// TIA Portal V20 export
DATA_BLOCK "InstShiftProductionTimes"   // DB113
TITLE = Instance ShiftProductionTimes
{ DB_Accessible_From_OPC_UA := 'FALSE' }
AUTHOR : SICAR
FAMILY : Shift
// Instance DB
// stored: DBAccessibleFromOPCUA false, InstanceOfName LSicar_ShiftProductionTimes, InstanceOfType FB
"LSicar_ShiftProductionTimes"
   // VAR_OUTPUT
   //    shiftProdTimeTarget { ExternalAccessible := 'False'; ExternalVisible := 'False'; ExternalWritable := 'False'} : Time := T#0MS;
   //    shiftProdTimeExpired { ExternalAccessible := 'False'; ExternalVisible := 'False'; ExternalWritable := 'False'} : Time := T#0MS;
   //    shiftActive { ExternalAccessible := 'False'; ExternalVisible := 'False'; ExternalWritable := 'False'} : Bool := FALSE;
   //    shiftFinishedPulse { ExternalAccessible := 'False'; ExternalVisible := 'False'; ExternalWritable := 'False'} : Bool := FALSE;
   // END_VAR
   // VAR_IN_OUT
   //    dateAndTime : "LSicar_typeGlobalDateTime";
   //    prodTimesHmi : "LSicar_typeProdTimesHmi";
   // END_VAR
   // VAR
   //    statCurrShiftTimes { ExternalAccessible := 'False'; ExternalVisible := 'False'; ExternalWritable := 'False'} : "LSicar_typeShiftTimes1Shift";
   //    statActual { ExternalAccessible := 'False'; ExternalVisible := 'False'; ExternalWritable := 'False'} : Time_Of_Day := TOD#00:00:00;
   //    statBefore { ExternalAccessible := 'False'; ExternalVisible := 'False'; ExternalWritable := 'False'} : Time_Of_Day := TOD#00:00:00;
   //    statDayChange { ExternalAccessible := 'False'; ExternalVisible := 'False'; ExternalWritable := 'False'} : Bool := FALSE;
   //    statDayChangeSet { ExternalAccessible := 'False'; ExternalVisible := 'False'; ExternalWritable := 'False'} : Bool := FALSE;
   //    statShift { ExternalAccessible := 'False'; ExternalVisible := 'False'; ExternalWritable := 'False'} : "LSicar_typeShiftmodelInfo";
   //    statProdTimeExpired { ExternalAccessible := 'False'; ExternalVisible := 'False'; ExternalWritable := 'False'} : Time := T#0MS;
   //    statBreak { ExternalAccessible := 'False'; ExternalVisible := 'False'; ExternalWritable := 'False'} : Array[0..4] of "LSicar_typeShiftmodelInfo";
   //    statBreakDurationSummary { ExternalAccessible := 'False'; ExternalVisible := 'False'; ExternalWritable := 'False'} : Time := T#0MS;
   //    statBreakActiveSummary { ExternalAccessible := 'False'; ExternalVisible := 'False'; ExternalWritable := 'False'} : Bool := FALSE;
   //    statBreakCount { ExternalAccessible := 'False'; ExternalVisible := 'False'; ExternalWritable := 'False'} : USInt := 0;
   //    statProdTimeExpired1 { ExternalAccessible := 'False'; ExternalVisible := 'False'; ExternalWritable := 'False'} : Time := T#0MS;
   //    statProdTimeExpired2 { ExternalAccessible := 'False'; ExternalVisible := 'False'; ExternalWritable := 'False'} : Time := T#0MS;
   //    statFalEdgeShiftActive { ExternalAccessible := 'False'; ExternalVisible := 'False'; ExternalWritable := 'False'} : Bool := FALSE;
   //    statNegPulseShiftActive { ExternalAccessible := 'False'; ExternalVisible := 'False'; ExternalWritable := 'False'} : Bool := FALSE;
   // END_VAR
BEGIN
   statCurrShiftTimes.start := TOD#00:00:00;
   statCurrShiftTimes.break[0..4].start := TOD#00:00:00;
   statCurrShiftTimes.break[0..4].startCircuitTime := TOD#00:00:00;
   statCurrShiftTimes.break[0..4].endCircuitTime := TOD#00:00:00;
   statCurrShiftTimes.break[0..4].end := TOD#00:00:00;
   statCurrShiftTimes.end := TOD#00:00:00;
   statShift.configured := FALSE;
   statShift.active := FALSE;
   statShift.duration := T#0MS;
   statBreak[0..4].configured := FALSE;
   statBreak[0..4].active := FALSE;
   statBreak[0..4].duration := T#0MS;
END_DATA_BLOCK
